FUNCTION_BLOCK FB_ControlSource_HMI EXTENDS FB_CyclicFB IMPLEMENTS I_PackML_ExternalController
VAR_INPUT
END_VAR

VAR_OUTPUT
END_VAR

VAR
	ipModule				  : I_PackML_Control;
	MainPMLControl_Simplified : ST_PackML_Control_Simplified;
	MainPMLControl_Standard	  : ST_PackML_Control;
	R_HMICommand			  : R_TRIG;
END_VAR

PROPERTY Control : SPT_BaseTypes.I_PackML_Control
SET
ipModule := Control;
END_SET
END_PROPERTY

METHOD CyclicLogic
VAR
	i : UDINT;
END_VAR
IF NOT _InitComplete THEN
	_InitComplete := Initialize();
	RETURN;
END_IF

MainPMLControl_Standard.CurrentMode	 := ipModule.CurrentMode;
MainPMLControl_Standard.CurrentState := ipModule.CurrentState;
FOR i := 1 TO 5 DO
	MainPMLControl_Standard.ModeNames[i] := F_UnitModeToString(UDINT_TO_DINT(i));
END_FOR

//Process HMI requests
R_HMICommand(CLK := (MainPMLControl_Simplified.ResetPressed XOR MainPMLControl_Simplified.StartPressed XOR MainPMLControl_Simplified.StopPressed) XOR (MainPMLControl_Standard.StateCommand <> E_PMLCommand.ePMLCommand_Undefined AND ipModule.StateCommand <> MainPMLControl_Standard.StateCommand) XOR (ipModule.ModeCommand <> MainPMLControl_Standard.ModeCommand));
IF R_HMICommand.Q THEN
	IF MainPMLControl_Simplified.ResetPressed AND MainPMLControl_Simplified.ResetPermissive AND MainPMLControl_Standard.CurrentState = E_PMLState.ePMLState_Aborted THEN
		ipModule.ChangeState(Tc3_PackML_V2.E_PMLCommand.ePMLCommand_Clear);
	ELSIF MainPMLControl_Simplified.ResetPressed AND MainPMLControl_Simplified.ResetPermissive THEN
		ipModule.ChangeState(Tc3_PackML_V2.E_PMLCommand.ePMLCommand_Reset);
	ELSIF MainPMLControl_Simplified.StartPressed AND MainPMLControl_Simplified.StartPermissive THEN
		IF MainPMLControl_Standard.CurrentState = Tc3_PackML_V2.E_PMLState.ePMLState_Idle THEN
			ipModule.ChangeState(Tc3_PackML_V2.E_PMLCommand.ePMLCommand_Start);
		ELSIF MainPMLControl_Standard.CurrentState = Tc3_PackML_V2.E_PMLState.ePMLState_Held THEN
			ipModule.ChangeState(Tc3_PackML_V2.E_PMLCommand.ePMLCommand_Unhold);
		END_IF
	ELSIF MainPMLControl_Simplified.StopPressed AND MainPMLControl_Simplified.StopPermissive THEN
		ipModule.ChangeState(Tc3_PackML_V2.E_PMLCommand.ePMLCommand_Stop);
	ELSIF ipModule.StateCommand <> MainPMLControl_Standard.StateCommand THEN
		ipModule.StateCommand := MainPMLControl_Standard.StateCommand;
	ELSIF ipModule.ModeCommand <> MainPMLControl_Standard.ModeCommand THEN
		ipModule.ModeCommand := MainPMLControl_Standard.ModeCommand;
	END_IF
END_IF

MainPMLControl_Simplified.StartPermissive := MainPMLControl_Standard.CurrentState = Tc3_PackML_V2.E_PMLState.ePMLState_Idle OR MainPMLControl_Standard.CurrentState = Tc3_PackML_V2.E_PMLState.ePMLState_Held;
MainPMLControl_Simplified.StopPermissive  := (MainPMLControl_Standard.CurrentState <> Tc3_PackML_V2.E_PMLState.ePMLState_Stopped AND MainPMLControl_Standard.CurrentState <> Tc3_PackML_V2.E_PMLState.ePMLState_Clearing AND MainPMLControl_Standard.CurrentState <> Tc3_PackML_V2.E_PMLState.ePMLState_Aborted AND MainPMLControl_Standard.CurrentState <> Tc3_PackML_V2.E_PMLState.ePMLState_Aborting AND
											  MainPMLControl_Standard.CurrentState <> Tc3_PackML_V2.E_PMLState.ePMLState_Undefined);

MainPMLControl_Simplified.ResetPermissive := MainPMLControl_Standard.CurrentState = Tc3_PackML_V2.E_PMLState.ePMLState_Complete OR MainPMLControl_Standard.CurrentState = Tc3_PackML_V2.E_PMLState.ePMLState_Stopped OR MainPMLControl_Standard.CurrentState = Tc3_PackML_V2.E_PMLState.ePMLState_Aborted;
END_METHOD

METHOD FINAL Initialize : BOOL
IF Registered THEN
	Initialize := TRUE;
END_IF
END_METHOD

METHOD FINAL ModeChanged
VAR_INPUT
	NewMode : SPT_BaseTypes.E_PMLUnitMode;
END_VAR
MainPMLControl_Standard.ModeCommand := NewMode;
END_METHOD

PROPERTY Registered : BOOL
GET
Registered := ipModule <> 0;
END_GET
END_PROPERTY

METHOD FINAL StateChanged
VAR_INPUT
	NewState : SPT_BaseTypes.E_PMLCommand;
END_VAR
MainPMLControl_Standard.StateCommand := NewState;
END_METHOD

END_FUNCTION_BLOCK

(* stored: Version 1.1.0.1, ProductVersion 3.1.4024.12
   POU FB_ControlSource_HMI: Id {13ebaa7c-af24-0bd6-2fec-aa1ce98efad0}, SpecialFunc None
   Folder I_CyclicFB: Id {da96ee3d-3a26-0760-3308-bd5f0e74cb8f}
   Folder I_PackML_ExternalController: Id {ee5784bf-99d0-0814-3e65-18ae759a9978}
   Property Control: Id {cce055b3-e7d5-0d5f-0873-78bf8c3fed60}
   Set Set: Id {baa4d435-ef43-0143-346d-f1ba06e17768}
   Method CyclicLogic: Id {44af9b85-e7ce-0cae-3b5b-4d8d8491eb58}
   Method Initialize: Id {f3e8687f-1037-0ff1-3a04-a5974da530c0}
   Method ModeChanged: Id {e837e8f8-b20d-086a-0e4c-5aefa38c717b}
   Property Registered: Id {bd443979-94b0-0160-3e10-60a25cf0cc83}
   Get Get: Id {1e227964-9dc4-00ac-0f7e-23b609f82ef8}
   Method StateChanged: Id {bb670118-8e4e-0208-05d7-955914bf17c7} *)
